INTERFACE I_Abortable EXTENDS __SYSTEM.IQueryInterface

METHOD Abort : HRESULT
VAR_INPUT
END_VAR
END_METHOD

END_INTERFACE

(* stored: Version 1.1.0.1
   Itf I_Abortable: Id {3a18816e-5c2a-4dda-91af-62fbcdd1161b}
   Method Abort: Id {17363283-e68f-4bd6-b67f-b264bff9b57d} *)
